// TIA Portal project "MPS_Sorting_mk3" (V16)

(* hardware
DEVICE "S7-1200 station_1"  S7-1200 Station
   slot 0: "Rack_0"  S7-1200 Rack  Rack  V1.0
   slot 1: "PLC_1"  CPU 1214C AC/DC/Rly  6ES7 214-1BG31-0XB0  V3.0
DEVICE "HMI_1"  KTP600 Basic color PN
   slot 0: "HMI_1"  KTP600 Basic color PN  6AV6 647-0AD11-3AX0  12.0.0.0
   slot 1: "HMI_RT_1"  KTP600 Basic color PN  6AV6 647-0AD11-3AX0  12.0.0.0
   slot 5: "HMI_1.IE_CP_1"  PROFINET Interface  12.0.0.0
      slot 1: "PROFINET Interface_1"  PROFINET Interface
         slot 1: "Port_1"  Port
*)

// ===== PLC "PLC_1"  CPU 1214C AC/DC/Rly =====

VAR_GLOBAL   // PLC tag table "Tabla de variables estándar"
   "Conveyor_Forward" AT %Q0.0 : Bool;
   "Extend_Def1" AT %Q0.1 : Bool;
   "Extend_Def2" AT %Q0.2 : Bool;
   "Retract_Stoper" AT %Q0.3 : Bool;
   "WP_at_Beg" AT %I0.0 : Bool;
   "Def1_Extended" AT %I0.1 : Bool;
   "Chute_Full" AT %I0.2 : Bool;
   "WP_Detected" AT %I0.4 : Bool;
   "WP_not_Black" AT %I0.5 : Bool;
   "WP_Metallic" AT %I0.6 : Bool;
   "System_Ready" AT %M0.0 : Bool;
   "Def2_Extended" AT %I0.3 : Bool;
   "WP_in_line" AT %M0.1 : Bool;
   "WP_at_Station" AT %M0.2 : Bool;
END_VAR

// folder: System blocks/Program resources

DATA_BLOCK "IEC_Timer_0_DB_2"   // DB2
{ S7_Optimized_Access := 'TRUE' }
AUTHOR : Simatic
FAMILY : IEC
NAME : IEC_TMR
VERSION : 1.0
// stored: InstanceOfName IEC_TIMER
"IEC_TIMER"
BEGIN
END_DATA_BLOCK

DATA_BLOCK "IEC_Timer_0_DB"   // DB3
{ S7_Optimized_Access := 'TRUE' }
AUTHOR : Simatic
FAMILY : IEC
NAME : IEC_TMR
VERSION : 1.0
// stored: InstanceOfName IEC_TIMER
"IEC_TIMER"
BEGIN
END_DATA_BLOCK

// folder: (top level)

FUNCTION "Op Main" : Void   // FC1, LAD
{ S7_Optimized_Access := 'TRUE' }
VERSION : 0.1
BEGIN

REGION Network 1: Banda Forward Inicial
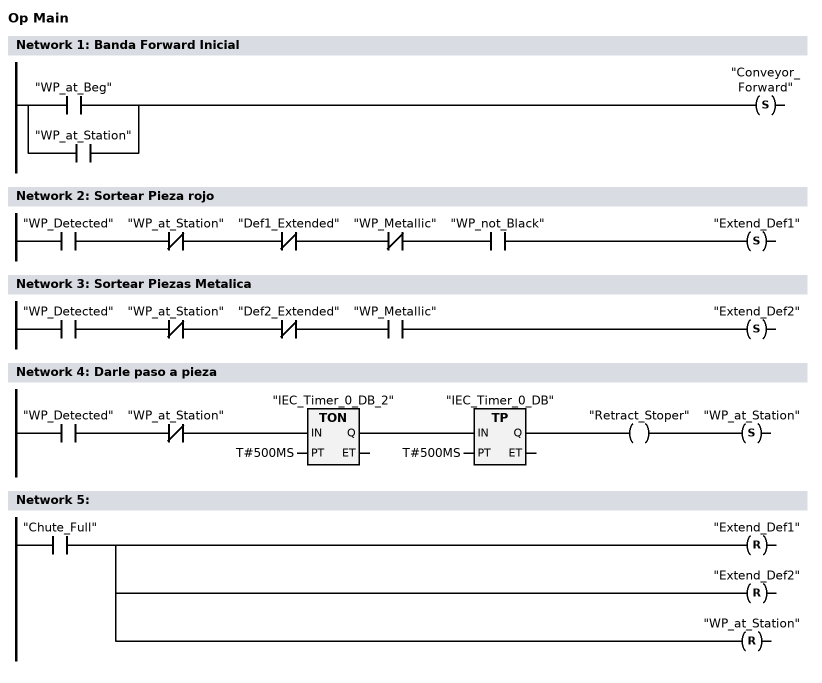
   RUNG wire#powerrail
      Contact( "WP_at_Beg" )
      wire#w1
      S_Coil( "Conveyor_Forward" )
   END_RUNG
   RUNG wire#powerrail
      Contact( "WP_at_Station" )
   END_RUNG wire#w1
   // the same network as SCL:
   IF "WP_at_Beg" OR "WP_at_Station" THEN "Conveyor_Forward" := TRUE; END_IF;
END_REGION

REGION Network 2: Sortear Pieza rojo
   RUNG wire#powerrail
      Contact( "WP_Detected" )
      I_Contact( "WP_at_Station" )
      I_Contact( "Def1_Extended" )
      I_Contact( "WP_Metallic" )
      Contact( "WP_not_Black" )
      S_Coil( "Extend_Def1" )
   END_RUNG
   // the same network as SCL:
   IF "WP_Detected" AND NOT "WP_at_Station" AND NOT "Def1_Extended" AND NOT "WP_Metallic" AND "WP_not_Black" THEN
       "Extend_Def1" := TRUE;
   END_IF;
END_REGION

REGION Network 3: Sortear Piezas Metalica
   RUNG wire#powerrail
      Contact( "WP_Detected" )
      I_Contact( "WP_at_Station" )
      I_Contact( "Def2_Extended" )
      Contact( "WP_Metallic" )
      S_Coil( "Extend_Def2" )
   END_RUNG
   // the same network as SCL:
   IF "WP_Detected" AND NOT "WP_at_Station" AND NOT "Def2_Extended" AND "WP_Metallic" THEN
       "Extend_Def2" := TRUE;
   END_IF;
END_REGION

REGION Network 4: Darle paso a pieza
   "IEC_Timer_0_DB_2".TON(IN := "WP_Detected" AND NOT "WP_at_Station", PT := T#500MS);
   "IEC_Timer_0_DB".TP(IN := "IEC_Timer_0_DB_2".Q, PT := T#500MS);
   "Retract_Stoper" := "IEC_Timer_0_DB".Q;
   IF "IEC_Timer_0_DB".Q THEN "WP_at_Station" := TRUE; END_IF;
END_REGION

REGION Network 5
   RUNG wire#powerrail
      Contact( "Chute_Full" )
      wire#w1
      R_Coil( "Extend_Def1" )
   END_RUNG
   RUNG wire#w1
      R_Coil( "Extend_Def2" )
   END_RUNG
   RUNG wire#w1
      R_Coil( "WP_at_Station" )
   END_RUNG
   // the same network as SCL:
   IF "Chute_Full" THEN
       "Extend_Def1" := FALSE;
       "Extend_Def2" := FALSE;
       "WP_at_Station" := FALSE;
   END_IF;
END_REGION
END_FUNCTION

ORGANIZATION_BLOCK "Main"   // OB1, LAD, ProgramCycle
TITLE = "Main Program Sweep (Cycle)"
{ S7_Optimized_Access := 'TRUE' }
VERSION : 0.1
BEGIN

REGION Network 1
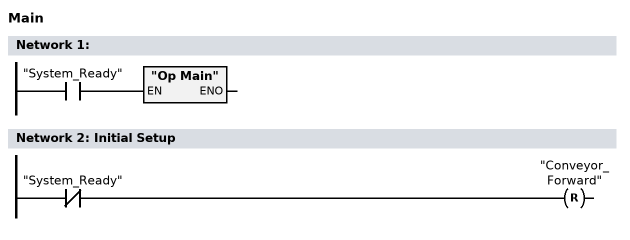
   RUNG wire#powerrail
      Contact( "System_Ready" )
      "Op Main"()
   END_RUNG
   // the same network as SCL:
   IF "System_Ready" THEN "Op Main"(); END_IF;
END_REGION

REGION Network 2: Initial Setup
   RUNG wire#powerrail
      I_Contact( "System_Ready" )
      R_Coil( "Conveyor_Forward" )
   END_RUNG
   // the same network as SCL:
   IF NOT "System_Ready" THEN "Conveyor_Forward" := FALSE; END_IF;
END_REGION
END_ORGANIZATION_BLOCK

ORGANIZATION_BLOCK "Startup"   // OB100, LAD, Startup
TITLE = "Complete Restart"
{ S7_Optimized_Access := 'TRUE' }
VERSION : 0.1
   VAR_INPUT
      LostRetentive : Bool;   // True if retentive data are lost
      LostRTC : Bool;   // True if date and time are lost
   END_VAR
BEGIN

REGION Network 1
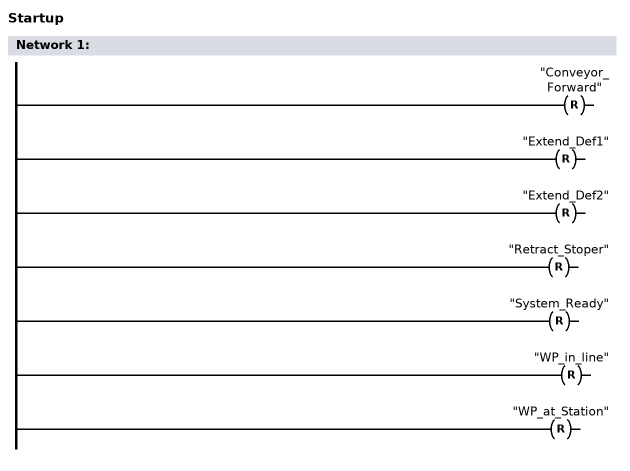
   RUNG wire#powerrail
      R_Coil( "Conveyor_Forward" )
   END_RUNG
   RUNG wire#powerrail
      R_Coil( "Extend_Def1" )
   END_RUNG
   RUNG wire#powerrail
      R_Coil( "Extend_Def2" )
   END_RUNG
   RUNG wire#powerrail
      R_Coil( "Retract_Stoper" )
   END_RUNG
   RUNG wire#powerrail
      R_Coil( "System_Ready" )
   END_RUNG
   RUNG wire#powerrail
      R_Coil( "WP_in_line" )
   END_RUNG
   RUNG wire#powerrail
      R_Coil( "WP_at_Station" )
   END_RUNG
   // the same network as SCL:
   "Conveyor_Forward" := FALSE;
   "Extend_Def1" := FALSE;
   "Extend_Def2" := FALSE;
   "Retract_Stoper" := FALSE;
   "System_Ready" := FALSE;
   "WP_in_line" := FALSE;
   "WP_at_Station" := FALSE;
END_REGION
END_ORGANIZATION_BLOCK

(* ===== HMI "HMI_RT_1" =====
system functions are stored by id; their names below are inferred from use
connection "HMI_Connection_1": ETHERNET, SMART_S7_1200_OMS

HMI tags "Default tag table"
   "Tag_ScreenNumber" : UInt, internal
   "System_Ready" : Bool = PLC System_Ready AT %M0.0, 1 s

Template "Template_1" 320x240
   Button "Exit" at 266,202 size 52x37; TextOff 'Exit'; PictureOff "ExitRuntime_KTP600_Basic_color_PN"; PictureOn "ExitRuntime_KTP600_Basic_color_PN"
      on Release: StopRuntime(0)
   Button "Template_Button" at 213,202 size 52x37; TextOff 'Text'
   Button "Template_Button_1" at 160,202 size 52x37; TextOff 'Text'
   Button "Template_Button_2" at 107,202 size 52x37; TextOff 'Text'
   Button "Alarms" at 54,202 size 52x37; TextOff 'Alarms'; PictureOff "AlarmDisplay_KTP600_Basic_color_PN"; PictureOn "AlarmDisplay_KTP600_Basic_color_PN"
      on Release: function_ef3f5d25("Alarm window_Unacknowledged", -1)
   Button "Start screen" at 1,202 size 52x37; TextOff 'Start screen'; PictureOff "NavigateHome_KTP600_Basic_color_PN"; PictureOn "NavigateHome_KTP600_Basic_color_PN"
      on Release: ActivateScreen("Root screen", 0)
   SymbolicIOField "Symbolic_IO_Field_Screen" at 69,7 size 164x24; TextOff '0'; TextOn '1'; TextList "TextList_ScreenNames"
      ProcessValue <- "Tag_ScreenNumber"
      on Change: ActivateScreenByNumber("Tag_ScreenNumber", 0)
   DateTimeField "HmiScreenItemData" at 235,19 size 85x19
   DateTimeField "HmiScreenItemData_1" at 235,0 size 85x19
   GraphicView "Logo" at 0,0 size 67x38; Picture "Logo of HMI_1"

screen "Root screen" 320x240, template "Template_1"
   on GenerateScreen: SetTag("Tag_ScreenNumber", 1)
   Button "Button_1" at 32,63 size 96x32; TextOff 'Start'
      on Press: SetBit("System_Ready")
   Button "Button_2" at 192,63 size 96x32; TextOff 'Stop'
      on Press: ResetBit("System_Ready")
   TextField "Text field_1" at 7,141 size 111x46; Text 'Por: Felipe Arenas Uribe Diego Lopez Guerrero Juan Pablo Tobos'
*)